(* IEC 61131-3 sources: cds-text-sync-reference-project/project-view/PLC/PLC Logic/FBD_Application/03_Object_POU_FBD/02_FunctionalBlock, 1 file *)

(* ---- FBD_FunctionBlock.ST_Method_under_XML.st ---- *)
METHOD ST_Method_under_XML : BOOL
VAR_INPUT
END_VAR

// --- implementation ---

ST_Method_under_XML := bool1 OR bool2;
//add comment123
